(*
    This test-suite runs several asserts with the same parameters (same expected, actual, message), calling the asserts
    in different cycles and using the same test.
    On top of this, we will call new asserts (though with same parameters) in later cycles.
    The reason we want the framework to support this is that theoretically the user could want to do an assert with the
    same message, using the same test with the same data values for both expected and actual, and splitting the asserts
    on different cycles.
*)
FUNCTION_BLOCK FB_AssertCountExceedsMaxNumber EXTENDS TcUnit.FB_TestSuite
VAR
END_VAR

Assert_SameEntryInOneCycle();
Assert_SameArrayEntryInOneCycle();

METHOD PRIVATE Assert_SameArrayEntryInOneCycle
VAR
    a : ARRAY[1..ArrayLength] OF DWORD := [16#12345678, 16#23456789];
    b : ARRAY[1..ArrayLength] OF DWORD := [16#90ABCDEF, 16#0ABCDEF1];
	
	i: UINT;
END_VAR
VAR CONSTANT
	ArrayLength : UINT := 2;
	MaxIndex : UINT := (TcUnit.GVL_Param_TcUnit.MaxNumberOfAssertsForEachTestSuite + 100); 
END_VAR
TEST('Assert_SameArrayEntryInOneCycle');

// Only checks if PLC crashes
FOR i := 1 TO MaxIndex DO
	AssertArrayEquals_DWORD(Expecteds := a,
						   	Actuals := a,
						   	Message := 'Values differ');
END_FOR;

AssertEquals_UINT(
		Expected:= GVL_Param_TcUnit.MaxNumberOfAssertsForEachTestSuite, 
		Actual:= AssertArrayResults.TotalArrayAsserts, 
		Message:= 'AssertArrayResults.TotalArrayAsserts invalid');

TEST_FINISHED();
END_METHOD

METHOD PRIVATE Assert_SameEntryInOneCycle
VAR
    a : DWORD := 16#12345678;
    b : DWORD := 16#90ABCDEF;
	
	i: UINT;
END_VAR
VAR CONSTANT
	MaxIndex : UINT := (TcUnit.GVL_Param_TcUnit.MaxNumberOfAssertsForEachTestSuite + 100); 
END_VAR
TEST('Assert_SameEntryInOneCycle');

// Only checks if PLC crashes
FOR i := 1 TO MaxIndex DO
	AssertEquals_DWORD(Expected := a,
					   Actual := a,
					   Message := 'Values differ');
END_FOR;

AssertEquals_UINT(
		Expected:= GVL_Param_TcUnit.MaxNumberOfAssertsForEachTestSuite, 
		Actual:= AssertResults.TotalAsserts, 
		Message:= 'AssertResults.TotalAsserts invalid');

TEST_FINISHED();
END_METHOD

END_FUNCTION_BLOCK

(* stored: Version 1.1.0.1, ProductVersion 3.1.4024.10
   POU FB_AssertCountExceedsMaxNumber: Id {5ccd4520-25c7-4bc8-a1a7-a6751f509f85}, SpecialFunc None
   Method Assert_SameArrayEntryInOneCycle: Id {6f972df2-c1ab-4b10-9350-030d31b8135f}
   Method Assert_SameEntryInOneCycle: Id {79d00f1b-a496-49a2-8093-dbe58274f7f4} *)
